(* IEC 61131-3 sources: Industry-PLC-LLM/data/PLCBEAD_repo/PLCBEAD_PLCEmbed-main/PLC-BEAD/Source/GEB/CSET, 1 file *)

(* ---- CSET.ST ---- *)
TYPE oscat_complex :
  STRUCT
	re : REAL;
	im : REAL;
  END_STRUCT;
END_TYPE

FUNCTION_BLOCK CSET_Block
	VAR_INPUT
		RE :	REAL;
		IM :	REAL;
	END_VAR

	VAR_OUTPUT
		CSET :	oscat_complex;
	END_VAR

	CSET.re := RE;
	CSET.im := IM;
END_FUNCTION_BLOCK

PROGRAM program0
  VAR
    LocalVar0 : REAL;
	LocalVaR1  : REAL;
	LocalOUT  : oscat_complex;
	func_block : CSET_Block;
  END_VAR
	func_block.RE  := LocalVar0;
	func_block.IM  := LocalVaR1 ;
	func_block();
	LocalOUT := func_block.CSET;
END_PROGRAM
